TYPE ST_OutputsMovableStop :
STRUCT
	HW					: ST_HW_OutputsMovableStop;		
END_STRUCT
END_TYPE

(* stored: Version 1.1.0.1, ProductVersion 3.1.4024.9
   DUT ST_OutputsMovableStop: Id {af97c1bf-35d0-4788-a81d-22c83ccfab0c} *)
